TYPE U_IN_IO_Translate :
UNION
	bArray :	ARRAY[1..32] OF BOOL;
	_Label :		INPUT_LABELS;
END_UNION
END_TYPE

(* stored: Version 1.1.0.1, ProductVersion 3.1.4024.10
   DUT U_IN_IO_Translate: Id {696a8959-8391-4850-a3b3-b2b5e52b1450} *)
